FUNCTION_BLOCK fbSCA
VAR_INPUT
	Interlock_1 : BOOL;
	Interlock_2 : BOOL;
	Interlock_3 : BOOL;
	Interlock_4 : BOOL;
	Interlock_5 : BOOL;
	Interlock_6 : BOOL;
	Interlock_7 : BOOL;
	
	AutoSP : REAL;
	CommandDirection : BOOL;
	AutoCmd : BOOL;
END_VAR
VAR_OUTPUT
	AutoMan : BOOL;
	ActualSpeed : REAL;
	ActualDirection : BOOL;
	Stopped : BOOL;
	Traveling : BOOL;
	Running : BOOL;
	Faulted : BOOL;
END_VAR
VAR
	StartCmdOut AT %Q* : BOOL;
	StopCmdOut AT %Q* : BOOL;
	Direction AT %Q* : BOOL;
	CommandSpeed : REAL;
	CommandSpeedRaw AT %Q* : DINT;
	ActualSpeedRaw AT %I*: DINT;
	Fault AT %I* : BOOL;
	EngMin : REAL := 0;		(* - means moving in the backward direction *)
	EngMax : REAL := 100;		(* the speed is expressed in percent *)
	RawMin : DINT := 2768;
	RawMax : DINT := 16535;
	Interlock_OK : BOOL;
	AutoReq : BOOL;
	ManReq : BOOL;
	ManSpeed : REAL;
	ManDirection : BOOL;
	ManStart : BOOL;
	ManStop : BOOL;

	strInterlock_1 : STRING;
	strInterlock_2 : STRING;
	strInterlock_3 : STRING;
	strInterlock_4 : STRING;
	strInterlock_5 : STRING;
	strInterlock_6 : STRING;
	strInterlock_7 : STRING;
	strAutoMan : STRING;
	idxStopTravRun : DINT;
	strStopTravRun : STRING;
	strOKFault : STRING;
	ClearFlt AT %Q* : BOOL;
	strAlmDesc : STRING;
	rCommandSpeed: REAL;		(* reserved variable *)
	
	simSCA : fbSimSCA;
	tmp: REAL;
END_VAR
VAR // added by the converter: edge detectors and wires of the graphical bodies
    _w1, _w2, _w3, _w4, _w5, _w6, _w7 : BOOL;
END_VAR

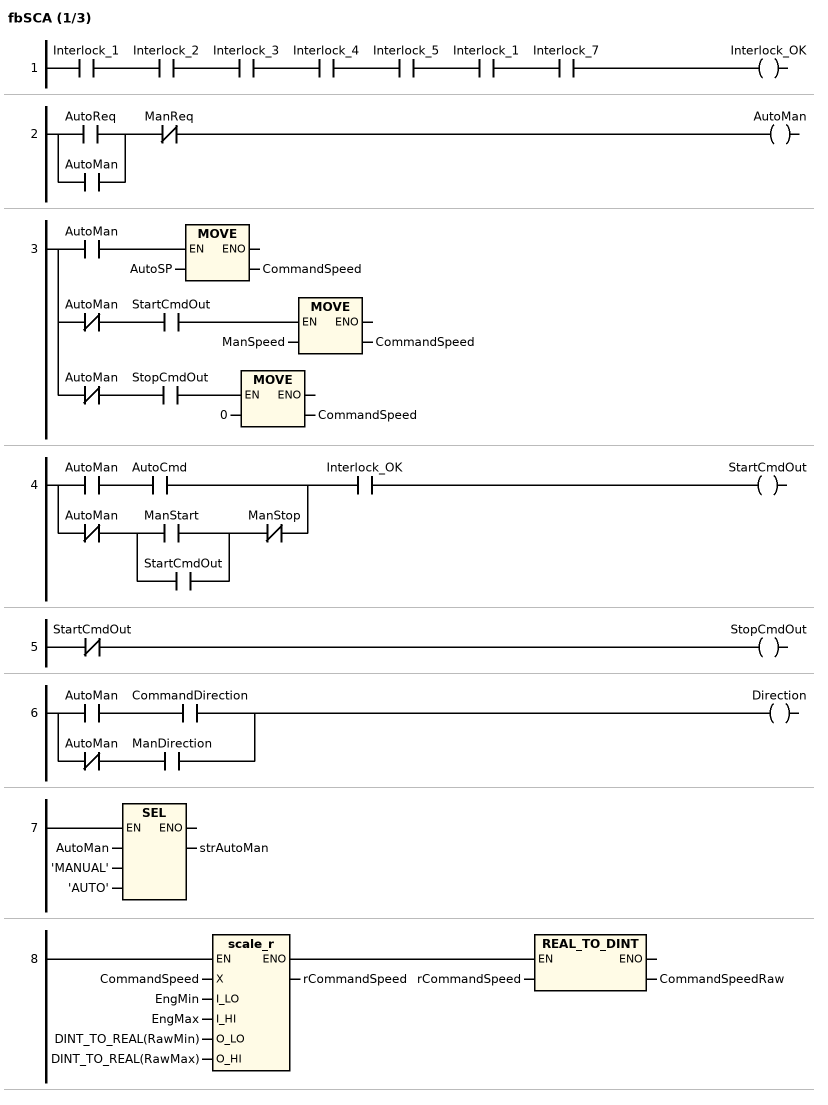
// NETWORK 1
Interlock_OK := Interlock_1 AND Interlock_2 AND Interlock_3 AND Interlock_4 AND Interlock_5 AND Interlock_1 AND Interlock_7;

// NETWORK 2
AutoMan := (AutoReq OR AutoMan) AND NOT ManReq;

// NETWORK 3
_w1 := AutoMan;
IF _w1 THEN CommandSpeed := AutoSP; END_IF
_w2 := NOT AutoMan AND StartCmdOut;
IF _w2 THEN CommandSpeed := ManSpeed; END_IF
_w3 := NOT AutoMan AND StopCmdOut;
IF _w3 THEN CommandSpeed := 0; END_IF
(* _w1 OR _w2 OR _w3; result not used *)

// NETWORK 4
StartCmdOut := (AutoMan AND AutoCmd OR NOT AutoMan AND (ManStart OR StartCmdOut) AND NOT ManStop) AND Interlock_OK;

// NETWORK 5
StopCmdOut := NOT StartCmdOut;

// NETWORK 6
Direction := AutoMan AND CommandDirection OR NOT AutoMan AND ManDirection;

// NETWORK 7
strAutoMan := SEL(AutoMan, 'MANUAL', 'AUTO');

// NETWORK 8
rCommandSpeed := scale_r(X := CommandSpeed, I_LO := EngMin, I_HI := EngMax, O_LO := DINT_TO_REAL(RawMin), O_HI := DINT_TO_REAL(RawMax));
CommandSpeedRaw := REAL_TO_DINT(rCommandSpeed);

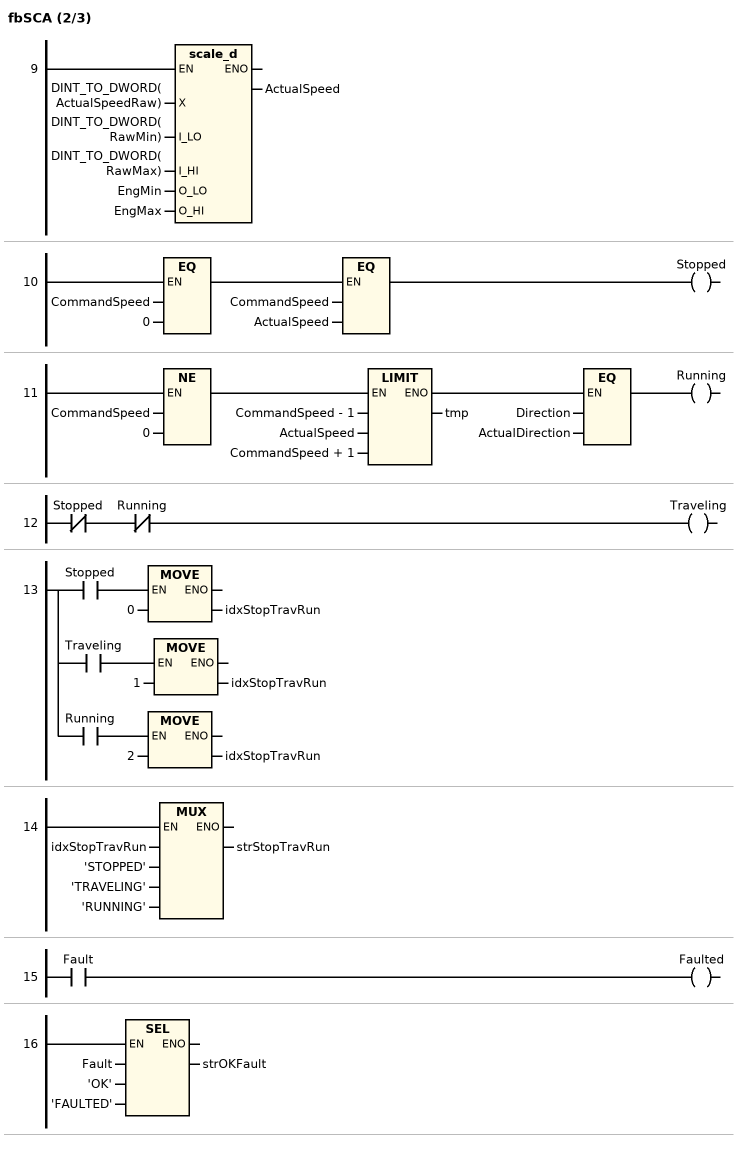
// NETWORK 9
ActualSpeed := scale_d(X := DINT_TO_DWORD(ActualSpeedRaw), I_LO := DINT_TO_DWORD(RawMin), I_HI := DINT_TO_DWORD(RawMax), O_LO := EngMin, O_HI := EngMax);

// NETWORK 10
Stopped := CommandSpeed = 0 AND CommandSpeed = ActualSpeed;

// NETWORK 11
_w4 := CommandSpeed <> 0;
IF _w4 THEN tmp := LIMIT(CommandSpeed - 1, ActualSpeed, CommandSpeed + 1); END_IF
Running := _w4 AND Direction = ActualDirection;

// NETWORK 12
Traveling := NOT Stopped AND NOT Running;

// NETWORK 13
_w5 := Stopped;
IF _w5 THEN idxStopTravRun := 0; END_IF
_w6 := Traveling;
IF _w6 THEN idxStopTravRun := 1; END_IF
_w7 := Running;
IF _w7 THEN idxStopTravRun := 2; END_IF
(* _w5 OR _w6 OR _w7; result not used *)

// NETWORK 14
strStopTravRun := MUX(idxStopTravRun, 'STOPPED', 'TRAVELING', 'RUNNING');

// NETWORK 15
Faulted := Fault;

// NETWORK 16
strOKFault := SEL(Fault, 'OK', 'FAULTED');

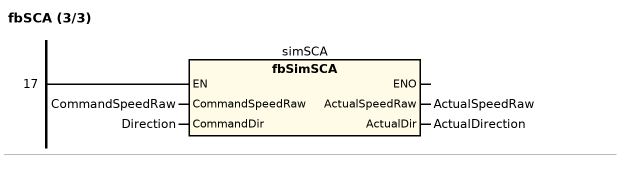
// NETWORK 17
simSCA(
    CommandSpeedRaw := CommandSpeedRaw,
    CommandDir := Direction,
    ActualSpeedRaw => ActualSpeedRaw,
    ActualDir => ActualDirection); // fbSimSCA

END_FUNCTION_BLOCK

(* stored: Version 1.1.0.1, ProductVersion 3.1.4022.17
   POU fbSCA: Id {86340b02-69fd-47a5-b7fb-abb2bd40ad59}, SpecialFunc None *)
